{attribute 'linkalways'} 
{attribute 'no_explicit_call' := 'This FB is a CLASS and must be accessed using methods or properties'}
{attribute 'enable_dynamic_creation'}
FUNCTION_BLOCK _TcVnVector3_UINT EXTENDS AliasDatatypeBase
VAR
	localData : TcVnVector3_UINT;
	activeData : REFERENCE TO TcVnVector3_UINT REF= localData;
	aliasBaseDatatype : _Array0to2OfUINT;
END_VAR

PROPERTY PUBLIC Address : PVOID
GET
Address := ADR(activeData);
END_GET
END_PROPERTY

METHOD PUBLIC ClearReference
VAR_INPUT
END_VAR
activeData REF= localData;
SetBaseDatatypeReference();
END_METHOD

METHOD PUBLIC Clone : I_Datatype
VAR
    pClone : POINTER TO _TcVnVector3_UINT;
END_VAR
pClone := __NEW(_TcVnVector3_UINT);
Clone := pClone^;
END_METHOD

METHOD FB_init : BOOL
VAR_INPUT
	bInitRetains : BOOL; // if TRUE, the retain variables are initialized (warm start / cold start)
	bInCopyCode : BOOL;  // if TRUE, the instance afterwards gets moved into the copy code (online change)
	//InitialValue : <type>; // if possible, not all values can be initialized
END_VAR
//localData := InitialValue; // if possible, not all values can be initialized
SetBaseDatatypeReference();
AddBaseDatatype(aliasBaseDatatype);
END_METHOD

PROPERTY PUBLIC Identifier : T_MAXSTRING
GET
Identifier := 'TcVnVector3_UINT';
END_GET
END_PROPERTY

METHOD PUBLIC MakeReferenceTo
VAR_INPUT
	ReferenceTarget : REFERENCE TO TcVnVector3_UINT;
END_VAR
activeData REF= ReferenceTarget;
SetBaseDatatypeReference();
END_METHOD

METHOD PROTECTED SetBaseDatatypeReference
VAR_INPUT
END_VAR
aliasBaseDatatype.MakeReferenceTo(activeData);
END_METHOD

PROPERTY PUBLIC Size : UDINT
GET
Size := SIZEOF(activeData);
END_GET
END_PROPERTY

METHOD TryMakeReferenceTo : BOOL
VAR_INPUT
	Target : I_Datatype;
END_VAR
VAR
	pTargetData : POINTER TO TcVnVector3_UINT;
END_VAR
IF NOT IsEquivalentTo(Target) THEN
	RETURN;
END_IF

pTargetData := Target.Address;
activeData REF= pTargetData^;
SetBaseDatatypeReference();
TryMakeReferenceTo := TRUE;
END_METHOD

PROPERTY PUBLIC Value : REFERENCE TO TcVnVector3_UINT
GET
Value REF= activeData;
END_GET
END_PROPERTY

END_FUNCTION_BLOCK

(* stored: Version 1.1.0.1, ProductVersion 3.1.4024.13
   POU _TcVnVector3_UINT: Id {c6ff79d9-3a8a-0f37-05ae-d588c6231896}, SpecialFunc None
   Folder Core: Id {235c60a2-a143-0262-217b-e52e4f49b4ac}
   Folder Protected: Id {7e72db0a-75ee-0aaa-173a-f96fe8b889d3}
   Folder Customize: Id {f0238811-702e-0151-1d77-1e2832340c5c}
   Folder Constructor: Id {25af080c-5221-0f45-3c5c-3aecf73b69b8}
   Property Address: Id {06c2433f-e025-07c5-0b9f-dd26778ec9a0}
   Get Get: Id {79fa2f9f-4a79-0398-30e4-79bbc6e438d2}
   Method ClearReference: Id {265346e0-1a3c-0e11-18eb-5871a615494d}
   Method Clone: Id {4f307ad8-e5c9-0325-0ae7-7faa7974d399}
   Method FB_init: Id {a6642e41-1f32-081b-1391-a09dc176ad0b}
   Property Identifier: Id {45fc912a-8bc1-0a01-1c9e-5d8f005959b6}
   Get Get: Id {a4b95aa2-38dc-0bbc-2c23-9cf06831df46}
   Method MakeReferenceTo: Id {67437477-39fd-03c6-1b71-2b8e7428edba}
   Method SetBaseDatatypeReference: Id {40cfcfff-e2e4-0364-0687-a2b0429d13aa}
   Property Size: Id {d61d0fa6-d0b2-0573-2632-57c7062ca5dc}
   Get Get: Id {7b427c31-421a-025f-3087-d6e0ce77d3cf}
   Method TryMakeReferenceTo: Id {cd49551f-26b8-006c-194e-e8e6cbdb05c3}
   Property Value: Id {8ddd8249-3e1f-0cfe-3ac2-3ff54997acd9}
   Get Get: Id {666846a8-7be5-099c-1844-078c82fd0c31} *)
